{attribute 'linkalways'} 
{attribute 'no_explicit_call' := 'This FB is a CLASS and must be accessed using methods or properties'}
{attribute 'enable_dynamic_creation'}
FUNCTION_BLOCK _ETcVnExtremePointDirection EXTENDS EnumDatatypeBase
VAR
	localData : ETcVnExtremePointDirection;
	activeData : REFERENCE TO ETcVnExtremePointDirection;
	enumBaseDatatype : _DINT(localData);
END_VAR

METHOD PRIVATE AddLocalEnumeration
VAR_INPUT
	Enumeration : T_MAXSTRING;
	Value : ETcVnExtremePointDirection;
END_VAR
AddEnumeration(Enumeration, Value);
END_METHOD

PROPERTY PUBLIC Address : PVOID
GET
Address := ADR(activeData);
END_GET
END_PROPERTY

METHOD PUBLIC ClearReference
VAR_INPUT
END_VAR
activeData REF= localData;
SetBaseDatatypeReference();
END_METHOD

METHOD PUBLIC Clone : I_Datatype
VAR
    pClone : POINTER TO _ETcVnExtremePointDirection;
END_VAR
pClone := __NEW(_ETcVnExtremePointDirection(InitialValue := Value));
Clone := pClone^;
END_METHOD

METHOD FB_init : BOOL
VAR_INPUT
	bInitRetains : BOOL; // if TRUE, the retain variables are initialized (warm start / cold start)
	bInCopyCode : BOOL;  // if TRUE, the instance afterwards gets moved into the copy code (online change)
	InitialValue : ETcVnExtremePointDirection;
END_VAR
localData := InitialValue;
AddBaseDatatype(enumBaseDatatype);
ClearReference();

AddLocalEnumeration('TCVN_EPD_TOP_LEFT', ETcVnExtremePointDirection.TCVN_EPD_TOP_LEFT);
AddLocalEnumeration('TCVN_EPD_TOP_MEDIAN', ETcVnExtremePointDirection.TCVN_EPD_TOP_MEDIAN);
AddLocalEnumeration('TCVN_EPD_TOP_RIGHT', ETcVnExtremePointDirection.TCVN_EPD_TOP_RIGHT);
AddLocalEnumeration('TCVN_EPD_BOTTOM_LEFT', ETcVnExtremePointDirection.TCVN_EPD_BOTTOM_LEFT);
AddLocalEnumeration('TCVN_EPD_BOTTOM_MEDIAN', ETcVnExtremePointDirection.TCVN_EPD_BOTTOM_MEDIAN);
AddLocalEnumeration('TCVN_EPD_BOTTOM_RIGHT', ETcVnExtremePointDirection.TCVN_EPD_BOTTOM_RIGHT);
AddLocalEnumeration('TCVN_EPD_LEFT_TOP', ETcVnExtremePointDirection.TCVN_EPD_LEFT_TOP);
AddLocalEnumeration('TCVN_EPD_LEFT_MEDIAN', ETcVnExtremePointDirection.TCVN_EPD_LEFT_MEDIAN);
AddLocalEnumeration('TCVN_EPD_LEFT_BOTTOM', ETcVnExtremePointDirection.TCVN_EPD_LEFT_BOTTOM);
AddLocalEnumeration('TCVN_EPD_RIGHT_TOP', ETcVnExtremePointDirection.TCVN_EPD_RIGHT_TOP);
AddLocalEnumeration('TCVN_EPD_RIGHT_MEDIAN', ETcVnExtremePointDirection.TCVN_EPD_RIGHT_MEDIAN);
AddLocalEnumeration('TCVN_EPD_RIGHT_BOTTOM', ETcVnExtremePointDirection.TCVN_EPD_RIGHT_BOTTOM);
END_METHOD

PROPERTY PUBLIC Identifier : T_MAXSTRING
GET
Identifier := 'ETcVnExtremePointDirection';
END_GET
END_PROPERTY

METHOD IsEnumeratorValueEqual : BOOL
VAR_INPUT
	Enumerator : I_KeyValueForwardEnumerator;
END_VAR
VAR
	storedValue : ETcVnExtremePointDirection;
END_VAR
IF NOT Enumerator.TryGet(storedValue) THEN
	RETURN;
END_IF

IsEnumeratorValueEqual := storedValue = activeData;
END_METHOD

METHOD PUBLIC MakeReferenceTo
VAR_INPUT
	ReferenceTarget : REFERENCE TO ETcVnExtremePointDirection;
END_VAR
activeData REF= ReferenceTarget;
SetBaseDatatypeReference();
END_METHOD

METHOD PROTECTED SetBaseDatatypeReference
VAR_INPUT
END_VAR
enumBaseDatatype.MakeReferenceTo(activeData);
END_METHOD

PROPERTY PUBLIC Size : UDINT
GET
Size := SIZEOF(activeData);
END_GET
END_PROPERTY

METHOD TryMakeReferenceTo : BOOL
VAR_INPUT
	Target : I_Datatype;
END_VAR
VAR
	targetAsEnum : I_EnumDatatype;
	pTargetData : POINTER TO ETcVnExtremePointDirection;
END_VAR
IF NOT Target.TryResolveAsEnumDatatype(targetAsEnum) THEN
	RETURN;
END_IF

IF targetAsEnum.Identifier <> Identifier THEN
	RETURN;
END_IF

pTargetData := Target.Address;
activeData REF= pTargetData^;
SetBaseDatatypeReference();
TryMakeReferenceTo := TRUE;
END_METHOD

PROPERTY PUBLIC Value : ETcVnExtremePointDirection
GET
Value := activeData;
END_GET
SET
activeData := Value;
END_SET
END_PROPERTY

END_FUNCTION_BLOCK

(* stored: Version 1.1.0.1
   POU _ETcVnExtremePointDirection: Id {581de72d-db94-4142-ab4f-76c109e3b1cf}, SpecialFunc None
   Folder Constructor: Id {19b9699b-d3ed-4c11-b9f2-20258e5c6cf6}
   Folder Private: Id {7e98bbff-217b-4651-b144-67640297998f}
   Folder Protected: Id {1f870cd8-1360-4b00-93a3-d0d7c6f6be7c}
   Method AddLocalEnumeration: Id {e8e30b0c-851c-4ef7-acf3-019dc7467a70}
   Property Address: Id {c5988636-2d63-46ef-925a-89f6d260e723}
   Get Get: Id {efa72679-3053-4d2f-b403-73bd974be70b}
   Method ClearReference: Id {72f0c32b-8915-4227-ac07-f2754af60300}
   Method Clone: Id {91d7c07f-1fde-4c80-9623-96f8c988208a}
   Method FB_init: Id {bcf3fc19-f6b3-4758-b6bb-adaf5b2b8953}
   Property Identifier: Id {8969303e-8a05-43df-aa6b-f04045b18f1e}
   Get Get: Id {01a32c03-20cd-405c-b536-c48b92ab3115}
   Method IsEnumeratorValueEqual: Id {3e2c9d7c-bd11-4fdf-bf7d-d168a655c3e5}
   Method MakeReferenceTo: Id {c5ea0db5-67b0-4a5c-9631-5599c54b9fa8}
   Method SetBaseDatatypeReference: Id {ef6e49fa-481d-4463-bbd5-bbc298ce4b12}
   Property Size: Id {b0b6c64d-9e76-4171-9aed-e809605a398b}
   Get Get: Id {a5d72a01-5326-42f2-9e9f-51f95f2312cd}
   Method TryMakeReferenceTo: Id {54d783dd-659a-44f5-90bc-980fde7f9856}
   Property Value: Id {fe4aa12d-d0b0-4a1f-8bdd-48a0ba8d6c43}
   Get Get: Id {6da81cd3-0ce0-48cd-99d8-e436642297cb}
   Set Set: Id {0fffa359-1f35-4c50-b49f-cac3a1b76ec8} *)
